// TIA Portal V20 export
FUNCTION_BLOCK "LER_thicknessHistory"   // FB71, LAD
// stored: Access Published, MemoryReserve 100, SetENOAutomatically false
   VAR_INPUT
      save_normal : Bool;
      "save_r&r" : Bool;
      result : "LER_typePartData";
   END_VAR
   VAR_IN_OUT
      dataHistory_normal : "LER_typeThicknessHistory";
      "dataHistory_r&r" : "LER_typeThicknessHistory_R&R";
   END_VAR
   VAR
      statDeleteData : "LER_typeThicknessHistory";
      statTrigger : Array[0..99] of Bool;
      statTonTimer : Array[0..99] of TON_TIME;
      statComplete : Array[0..99] of Bool;
   END_VAR
   VAR_TEMP
      tempRetVal : Array[0..99] of Int;
   END_VAR
   VAR_TEMP   // added for the SCL form of the ladder/FBD networks
      _w1 : Bool;
   END_VAR
BEGIN

REGION Network 1: NORMAL
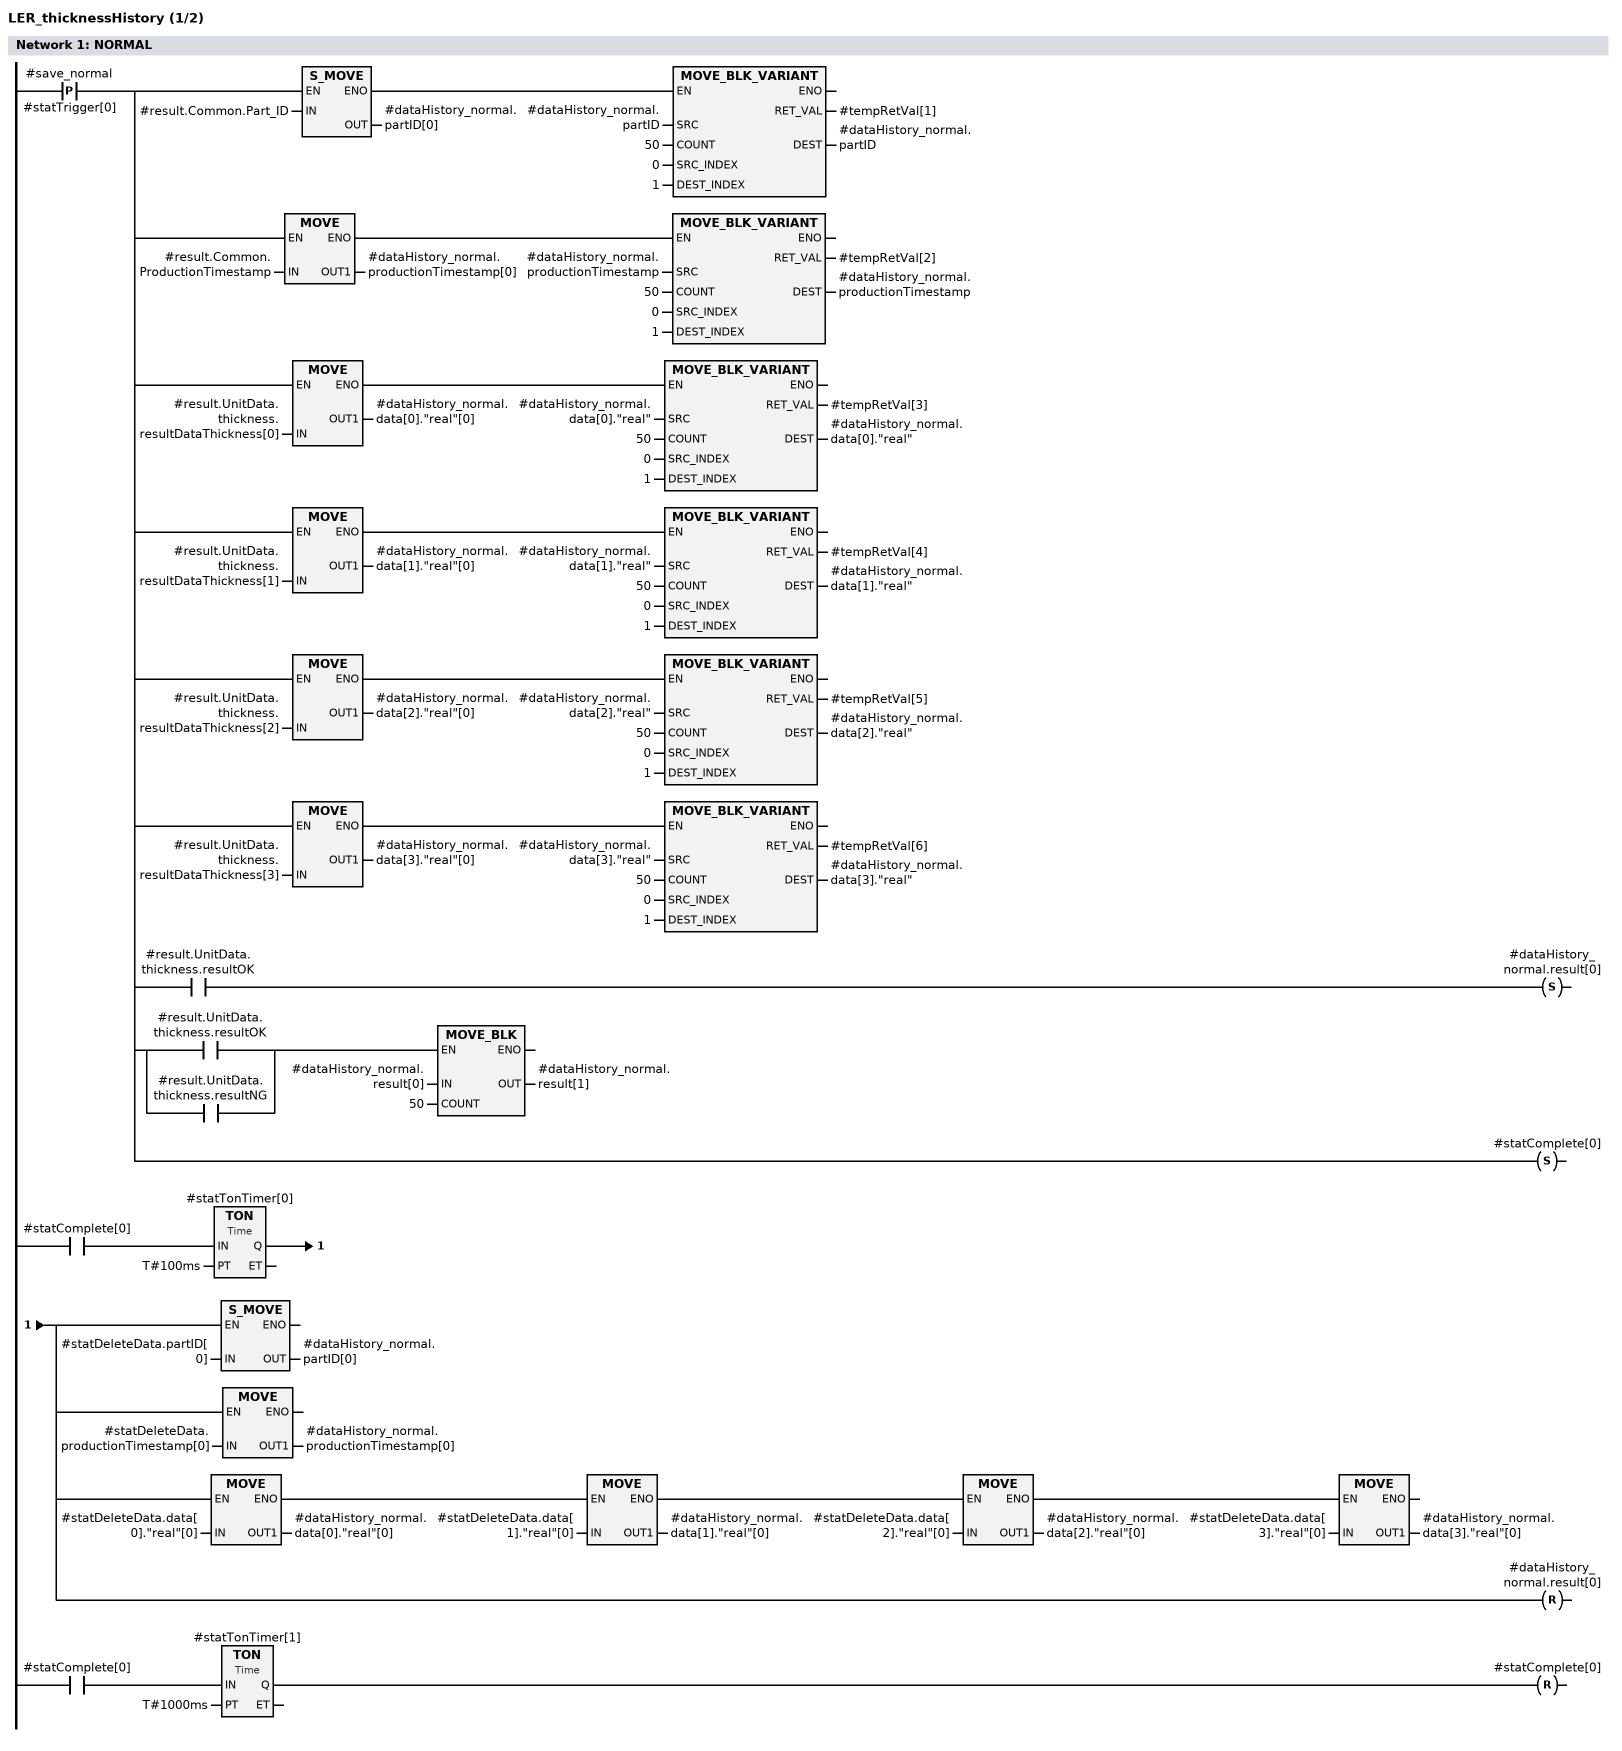
   #_w1 := #save_normal AND NOT #statTrigger[0];   // rising edge of #save_normal
   #statTrigger[0] := #save_normal;
   IF #_w1 THEN
       #dataHistory_normal.partID[0] := #result.Common.Part_ID;
       #tempRetVal[1] := MOVE_BLK_VARIANT(SRC := #dataHistory_normal.partID,
                               COUNT := 50,
                               SRC_INDEX := 0,
                               DEST_INDEX := 1,
                               DEST => #dataHistory_normal.partID);
       #dataHistory_normal.productionTimestamp[0] := #result.Common.ProductionTimestamp;
       #tempRetVal[2] := MOVE_BLK_VARIANT(SRC := #dataHistory_normal.productionTimestamp,
                               COUNT := 50,
                               SRC_INDEX := 0,
                               DEST_INDEX := 1,
                               DEST => #dataHistory_normal.productionTimestamp);
       #dataHistory_normal.data[0]."real"[0] := #result.UnitData.thickness.resultDataThickness[0];
       #tempRetVal[3] := MOVE_BLK_VARIANT(SRC := #dataHistory_normal.data[0]."real",
                               COUNT := 50,
                               SRC_INDEX := 0,
                               DEST_INDEX := 1,
                               DEST => #dataHistory_normal.data[0]."real");
       #dataHistory_normal.data[1]."real"[0] := #result.UnitData.thickness.resultDataThickness[1];
       #tempRetVal[4] := MOVE_BLK_VARIANT(SRC := #dataHistory_normal.data[1]."real",
                               COUNT := 50,
                               SRC_INDEX := 0,
                               DEST_INDEX := 1,
                               DEST => #dataHistory_normal.data[1]."real");
       #dataHistory_normal.data[2]."real"[0] := #result.UnitData.thickness.resultDataThickness[2];
       #tempRetVal[5] := MOVE_BLK_VARIANT(SRC := #dataHistory_normal.data[2]."real",
                               COUNT := 50,
                               SRC_INDEX := 0,
                               DEST_INDEX := 1,
                               DEST => #dataHistory_normal.data[2]."real");
       #dataHistory_normal.data[3]."real"[0] := #result.UnitData.thickness.resultDataThickness[3];
       #tempRetVal[6] := MOVE_BLK_VARIANT(SRC := #dataHistory_normal.data[3]."real",
                               COUNT := 50,
                               SRC_INDEX := 0,
                               DEST_INDEX := 1,
                               DEST => #dataHistory_normal.data[3]."real");
   END_IF;
   IF #_w1 AND #result.UnitData.thickness.resultOK THEN #dataHistory_normal.result[0] := TRUE; END_IF;
   IF #_w1 AND (#result.UnitData.thickness.resultOK OR #result.UnitData.thickness.resultNG) THEN
       MOVE_BLK(IN := #dataHistory_normal.result[0], COUNT := 50, OUT => #dataHistory_normal.result[1]);
   END_IF;
   IF #_w1 THEN #statComplete[0] := TRUE; END_IF;
   #statTonTimer[0].TON(IN := #statComplete[0], PT := T#100ms);
   IF #statTonTimer[0].Q THEN
       #dataHistory_normal.partID[0] := #statDeleteData.partID[0];
       #dataHistory_normal.productionTimestamp[0] := #statDeleteData.productionTimestamp[0];
       #dataHistory_normal.data[0]."real"[0] := #statDeleteData.data[0]."real"[0];
       #dataHistory_normal.data[1]."real"[0] := #statDeleteData.data[1]."real"[0];
       #dataHistory_normal.data[2]."real"[0] := #statDeleteData.data[2]."real"[0];
       #dataHistory_normal.data[3]."real"[0] := #statDeleteData.data[3]."real"[0];
       #dataHistory_normal.result[0] := FALSE;
   END_IF;
   #statTonTimer[1].TON(IN := #statComplete[0], PT := T#1000ms);
   IF #statTonTimer[1].Q THEN #statComplete[0] := FALSE; END_IF;
END_REGION

REGION Network 2: R&R
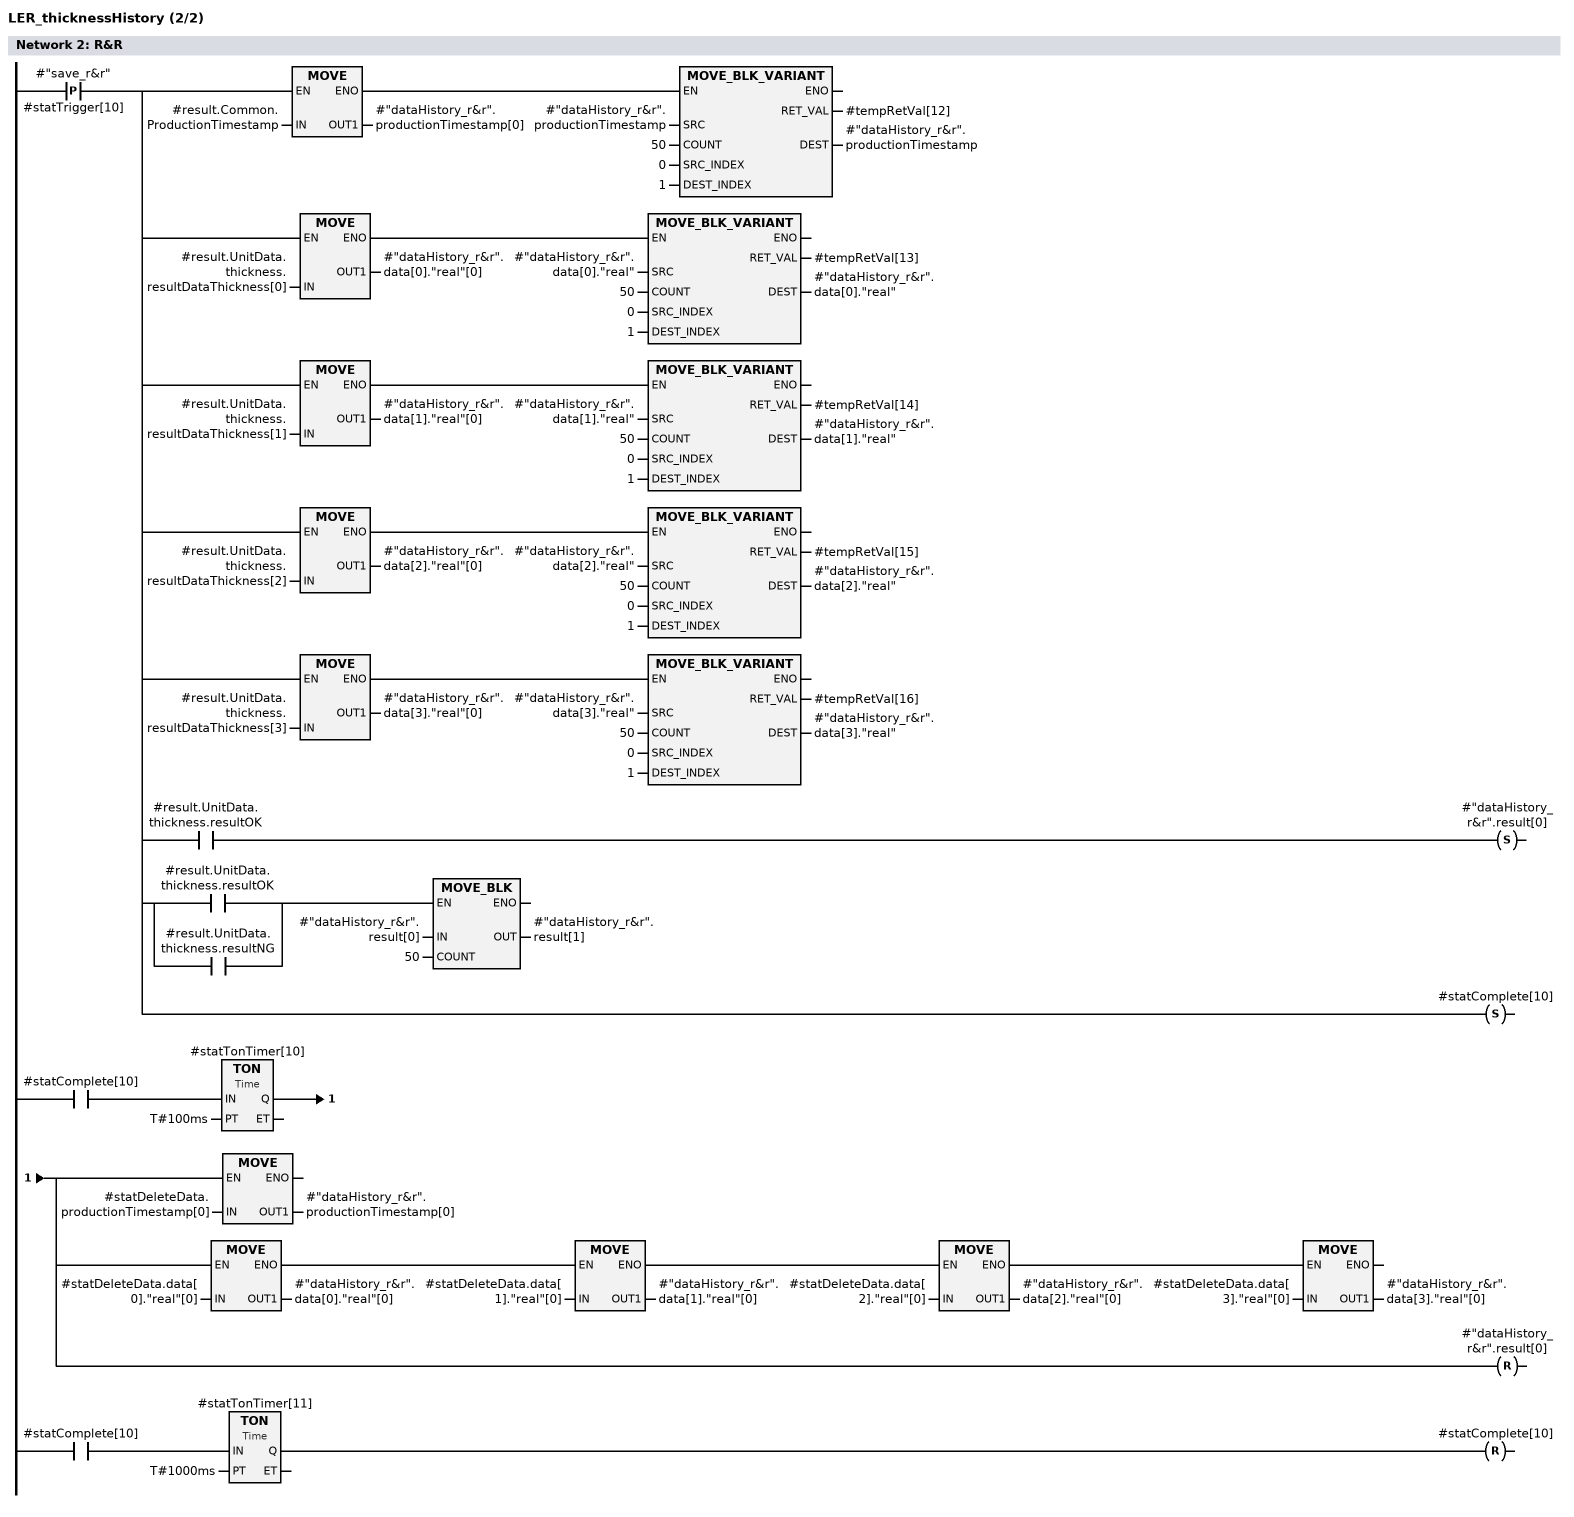
   #_w1 := #"save_r&r" AND NOT #statTrigger[10];   // rising edge of #"save_r&r"
   #statTrigger[10] := #"save_r&r";
   IF #_w1 THEN
       #"dataHistory_r&r".productionTimestamp[0] := #result.Common.ProductionTimestamp;
       #tempRetVal[12] := MOVE_BLK_VARIANT(SRC := #"dataHistory_r&r".productionTimestamp,
                               COUNT := 50,
                               SRC_INDEX := 0,
                               DEST_INDEX := 1,
                               DEST => #"dataHistory_r&r".productionTimestamp);
       #"dataHistory_r&r".data[0]."real"[0] := #result.UnitData.thickness.resultDataThickness[0];
       #tempRetVal[13] := MOVE_BLK_VARIANT(SRC := #"dataHistory_r&r".data[0]."real",
                               COUNT := 50,
                               SRC_INDEX := 0,
                               DEST_INDEX := 1,
                               DEST => #"dataHistory_r&r".data[0]."real");
       #"dataHistory_r&r".data[1]."real"[0] := #result.UnitData.thickness.resultDataThickness[1];
       #tempRetVal[14] := MOVE_BLK_VARIANT(SRC := #"dataHistory_r&r".data[1]."real",
                               COUNT := 50,
                               SRC_INDEX := 0,
                               DEST_INDEX := 1,
                               DEST => #"dataHistory_r&r".data[1]."real");
       #"dataHistory_r&r".data[2]."real"[0] := #result.UnitData.thickness.resultDataThickness[2];
       #tempRetVal[15] := MOVE_BLK_VARIANT(SRC := #"dataHistory_r&r".data[2]."real",
                               COUNT := 50,
                               SRC_INDEX := 0,
                               DEST_INDEX := 1,
                               DEST => #"dataHistory_r&r".data[2]."real");
       #"dataHistory_r&r".data[3]."real"[0] := #result.UnitData.thickness.resultDataThickness[3];
       #tempRetVal[16] := MOVE_BLK_VARIANT(SRC := #"dataHistory_r&r".data[3]."real",
                               COUNT := 50,
                               SRC_INDEX := 0,
                               DEST_INDEX := 1,
                               DEST => #"dataHistory_r&r".data[3]."real");
   END_IF;
   IF #_w1 AND #result.UnitData.thickness.resultOK THEN #"dataHistory_r&r".result[0] := TRUE; END_IF;
   IF #_w1 AND (#result.UnitData.thickness.resultOK OR #result.UnitData.thickness.resultNG) THEN
       MOVE_BLK(IN := #"dataHistory_r&r".result[0], COUNT := 50, OUT => #"dataHistory_r&r".result[1]);
   END_IF;
   IF #_w1 THEN #statComplete[10] := TRUE; END_IF;
   #statTonTimer[10].TON(IN := #statComplete[10], PT := T#100ms);
   IF #statTonTimer[10].Q THEN
       #"dataHistory_r&r".productionTimestamp[0] := #statDeleteData.productionTimestamp[0];
       #"dataHistory_r&r".data[0]."real"[0] := #statDeleteData.data[0]."real"[0];
       #"dataHistory_r&r".data[1]."real"[0] := #statDeleteData.data[1]."real"[0];
       #"dataHistory_r&r".data[2]."real"[0] := #statDeleteData.data[2]."real"[0];
       #"dataHistory_r&r".data[3]."real"[0] := #statDeleteData.data[3]."real"[0];
       #"dataHistory_r&r".result[0] := FALSE;
   END_IF;
   #statTonTimer[11].TON(IN := #statComplete[10], PT := T#1000ms);
   IF #statTonTimer[11].Q THEN #statComplete[10] := FALSE; END_IF;
END_REGION
END_FUNCTION_BLOCK
